FUNCTION_BLOCK AX_X_TO_BOOL (* Composite FB for convert AX to BOOL *)
  (* Standard: 61499-2 *)
  (* Version 1.0, 2024-04-24, franz *)
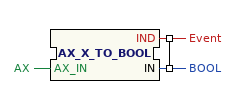
  EVENT_OUTPUT
    IND WITH IN; (* Initialization Confirm *)
  END_EVENT
  VAR_OUTPUT
    IN : BOOL;
  END_VAR
  SOCKETS
    AX_IN : AX;
  END_SOCKETS
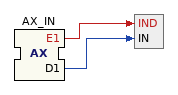
  EVENT_CONNECTIONS
    AX_IN.E1 TO IND;
  END_CONNECTIONS
  DATA_CONNECTIONS
    AX_IN.D1 TO IN;
  END_CONNECTIONS
END_FUNCTION_BLOCK
